// TIA Portal V16 export
// export: Created 2022-12-22T10:22:46.3749075Z, ExportSetting WithDefaults, DisplayName Totally Integrated Automation Portal, DisplayVersion V16, DisplayName TIA Portal Version Control Interface, DisplayVersion V16, DisplayName TIA Portal Openness, DisplayVersion V16, DisplayName STEP 7 Professional, DisplayVersion V16, DisplayName STEP 7 Safety, DisplayVersion V16, DisplayName WinCC Advanced, DisplayVersion V16
ORGANIZATION_BLOCK "Main"   // OB1, LAD, ProgramCycle
TITLE = "Main Program Sweep (Cycle)"
{ S7_Optimized_Access := 'TRUE' }
VERSION : 0.1
// stored: AutoNumber true, IsIECCheckEnabled false, SetENOAutomatically false
   VAR_INPUT
      Initial_Call : Bool;   // Initial call of this OB
      Remanence : Bool;   // =True, if remanent data are available
   END_VAR
BEGIN

REGION Network 1
   // test demo - v1
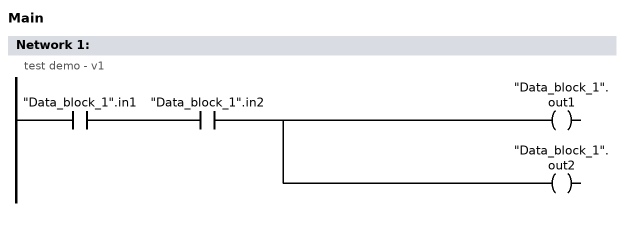
   RUNG wire#powerrail
      Contact( "Data_block_1".in1 )
      Contact( "Data_block_1".in2 )
      wire#w1
      Coil( "Data_block_1".out1 )
   END_RUNG
   RUNG wire#w1
      Coil( "Data_block_1".out2 )
   END_RUNG
   // the same network as SCL:
   "Data_block_1".out1 := "Data_block_1".in1 AND "Data_block_1".in2;
   "Data_block_1".out2 := "Data_block_1".out1;
END_REGION
END_ORGANIZATION_BLOCK
